IF st_config.b_config_fertig THEN
	(* Fehlermeldungen und Betriebsmeldungen ab dem Startindex in die globalen Meldungsarrays schreiben *)
	garr_stoermeldungen[st_config.i16_meld_startindex + 0] := sm_haspel_notaus;
	garr_stoermeldungen[st_config.i16_meld_startindex + 1] := sm_haspel_notabschaltung;
	garr_stoermeldungen[st_config.i16_meld_startindex + 2] := FALSE;
	garr_stoermeldungen[st_config.i16_meld_startindex + 3] := FALSE;
	garr_stoermeldungen[st_config.i16_meld_startindex + 4] := FALSE;
	garr_stoermeldungen[st_config.i16_meld_startindex + 5] := FALSE;
	garr_stoermeldungen[st_config.i16_meld_startindex + 6] := FALSE;
	garr_stoermeldungen[st_config.i16_meld_startindex + 7] := FALSE;
	garr_stoermeldungen[st_config.i16_meld_startindex + 8] := FALSE;
	garr_stoermeldungen[st_config.i16_meld_startindex + 9] := FALSE;
	garr_stoermeldungen[st_config.i16_meld_startindex + 10] := FALSE;
	garr_stoermeldungen[st_config.i16_meld_startindex + 11] := FALSE;
	garr_stoermeldungen[st_config.i16_meld_startindex + 12] := FALSE;
	garr_stoermeldungen[st_config.i16_meld_startindex + 13] := FALSE;
	garr_stoermeldungen[st_config.i16_meld_startindex + 14] := FALSE;
	garr_stoermeldungen[st_config.i16_meld_startindex + 15] := FALSE;
	garr_stoermeldungen[st_config.i16_meld_startindex + 16] := FALSE;
	garr_stoermeldungen[st_config.i16_meld_startindex + 17] := FALSE;
	garr_stoermeldungen[st_config.i16_meld_startindex + 18] := FALSE;
	garr_stoermeldungen[st_config.i16_meld_startindex + 19] := FALSE;
	
	garr_betriebsmeldungen[st_config.i16_meld_startindex + 0] := bm_haspel_bandende;
	garr_betriebsmeldungen[st_config.i16_meld_startindex + 1] := FALSE;
	garr_betriebsmeldungen[st_config.i16_meld_startindex + 2] := FALSE;
	garr_betriebsmeldungen[st_config.i16_meld_startindex + 3] := FALSE;
	garr_betriebsmeldungen[st_config.i16_meld_startindex + 4] := FALSE;
	garr_betriebsmeldungen[st_config.i16_meld_startindex + 5] := FALSE;
	garr_betriebsmeldungen[st_config.i16_meld_startindex + 6] := FALSE;
	garr_betriebsmeldungen[st_config.i16_meld_startindex + 7] := FALSE;
	garr_betriebsmeldungen[st_config.i16_meld_startindex + 8] := FALSE;
	garr_betriebsmeldungen[st_config.i16_meld_startindex + 9] := FALSE;
	garr_betriebsmeldungen[st_config.i16_meld_startindex + 10] := FALSE;
	garr_betriebsmeldungen[st_config.i16_meld_startindex + 11] := FALSE;
	garr_betriebsmeldungen[st_config.i16_meld_startindex + 12] := FALSE;
	garr_betriebsmeldungen[st_config.i16_meld_startindex + 13] := FALSE;
	garr_betriebsmeldungen[st_config.i16_meld_startindex + 14] := FALSE;
	garr_betriebsmeldungen[st_config.i16_meld_startindex + 15] := FALSE;
	garr_betriebsmeldungen[st_config.i16_meld_startindex + 16] := FALSE;
	garr_betriebsmeldungen[st_config.i16_meld_startindex + 17] := FALSE;
	garr_betriebsmeldungen[st_config.i16_meld_startindex + 18] := FALSE;
	garr_betriebsmeldungen[st_config.i16_meld_startindex + 19] := FALSE;
END_IF
END_FUNCTION_BLOCK

(* POU Gemeinsamkeiten17xx/Oeler/ST_Bandoeler, ST *)
FUNCTION_BLOCK ST_Bandoeler
VAR_INPUT
	st_config						: struct_config;
	st_ctrl_in						: struct_ctrl_in;
	b_ot_spur					: BOOL;
END_VAR
VAR_IN_OUT
	st_daten						: struct_oeler_daten;
	st_visu						: struct_oeler_visu;
END_VAR
VAR_OUTPUT
	st_ctrl_out					: struct_ctrl_out;
END_VAR
VAR
	fb_ton_quitt					: TON;
	dt_datum_uhrzeit_letzte_oelung	: DT;
	fb_state_entry					: ST_StateEntry;
	t_delta_zeitraum				: TIME := t#5h;
	t_blaszeit					: TIME := t#500ms;
	fb_ton_oelzeit					: TON;
	fb_ton_blaszeit				: TON;
	fb_r_trig_start_oelen			: R_TRIG;
	fb_r_trig_hubimpuls			: R_TRIG;
	i32_default_wert_intervall		: INT := 1000;

	fb_r_trig_ibn_handoelen		: R_TRIG;
	fb_ton_ibn_handoelen			: TON;
	b_ibn_handoelen				: BOOL := FALSE;

	a_ventil_oel		 			AT %Q* : BOOL;
	a_ventil_luft		 			AT %Q* : BOOL;
END_VAR
(* Bandöler mit Zwangs- und Stillstandsölung *)
(* Oeler Impuls generieren *)
fb_ton_oelzeit(IN:= , PT:= , Q=> , ET=> );
fb_ton_blaszeit(IN:= , PT:= t_blaszeit, Q=> , ET=> );
fb_ton_quitt(IN:= , PT:= t#100ms, Q=> , ET=> );

(* Hubimpuls *)
fb_r_trig_hubimpuls(CLK:= b_ot_spur, Q=> );

(* Inbetriebnahme *)
fb_r_trig_ibn_handoelen(CLK:= b_ibn_handoelen, Q=> );
fb_ton_ibn_handoelen(IN:= , PT:= t#1s, Q=> , ET=> );
IF fb_r_trig_ibn_handoelen.Q THEN
	fb_ton_ibn_handoelen.IN := TRUE;
ELSE
	IF fb_ton_ibn_handoelen.Q THEN
		b_ibn_handoelen := FALSE;
	 	fb_ton_ibn_handoelen.IN := FALSE;
	END_IF
END_IF

(* =======================================Toplevel========================================== *)
IF fb_state_entry.i16_next_step > INIT AND fb_state_entry.i16_next_step < FEHLER THEN
	IF fb_state_entry.i16_next_step < STOP THEN
		IF st_ctrl_in.b_stop THEN
			fb_state_entry.i16_next_step := STOP;
		END_IF
	END_IF
END_IF

(* Prüfe auf neue Intervalvorgabe *)
IF st_config.b_station_aktiv AND st_daten.i32_neue_intervallvorgabe <> st_daten.i32_alte_intervallvorgabe THEN
	st_daten.i32_alte_intervallvorgabe := st_daten.i32_neue_intervallvorgabe;
	st_daten.i32_aktueller_stand := st_daten.i32_neue_intervallvorgabe;
END_IF

(* Zähle Hübe *)
IF st_config.b_station_aktiv AND fb_r_trig_hubimpuls.Q THEN
	(* Von der Intervallvorgabe wird runter gezählt bis Null. Dann kommt der Ölimpuls *)
	st_daten.i32_aktueller_stand := st_daten.i32_aktueller_stand - 1;
END_IF

(* ==================================Schrittkette================================ *)
fb_state_entry(
	i16_next_step:= , 
	i16_pos:= 1,
	s_debugtext:= ,
	E=> ,
	X=> , 
	i16_step=> ,
	i16_last_step=> );

CASE fb_state_entry.i16_step OF
(*=======================================================*)
	INIT_OBJ:
		IF st_config.b_config_fertig THEN
			fb_state_entry.i16_next_step := INIT;
		END_IF
		
(*=======================================================*)
	INIT:
		IF fb_state_entry.E THEN
			fb_ton_blaszeit.IN := FALSE;
			fb_ton_oelzeit.IN := FALSE;
			st_ctrl_out.b_fehler := FALSE;
			st_ctrl_out.b_bereit := FALSE;
			st_ctrl_out.b_fertig := FALSE;
			a_ventil_oel := FALSE;
			a_ventil_luft := FALSE;
		END_IF

		(*-----------------------Weiterschaltbedingungen----------------------------*)
		IF st_ctrl_in.b_init THEN
			IF st_config.b_station_aktiv THEN
				fb_state_entry.i16_next_step := 20;
			ELSE
				fb_state_entry.i16_next_step := BEREIT;
			END_IF
		END_IF

(*=======================================================*)
	20: (* Abfrage Datum / Uhrzeit wegen Ölen nach Stillstand*)

		(*-----------------------Weiterschaltbedingungen----------------------------*)
		IF (gdt_system_time - dt_datum_uhrzeit_letzte_oelung) > t_delta_zeitraum THEN
			fb_ton_oelzeit.PT := st_daten.t_oelzeit_nach_stillstand;
			fb_state_entry.i16_next_step := 110;
		ELSE
			fb_state_entry.i16_next_step := BEREIT;
		END_IF

(*=======================================================*)
	BEREIT:
		IF fb_state_entry.E THEN
			st_ctrl_out.b_bereit := TRUE;
		END_IF

		(*-----------------------Weiterschaltbedingungen----------------------------*)
		IF  st_config.b_station_aktiv AND (st_daten.i32_aktueller_stand <= 0 OR st_visu.b_handoelen OR fb_r_trig_ibn_handoelen.Q) THEN
			st_visu.b_handoelen := FALSE;
			fb_ton_oelzeit.PT := st_daten.t_ventiloeffnungszeit;
			fb_state_entry.i16_next_step := 110;
		END_IF

(*=======================================================*)
	110: (* Luft einschalten *)
		IF fb_state_entry.E THEN
			fb_ton_blaszeit.IN := TRUE;
			a_ventil_luft := TRUE;
		END_IF

		(*-----------------------Weiterschaltbedingungen----------------------------*)
		IF  fb_ton_blaszeit.Q THEN
			fb_ton_blaszeit.IN := FALSE;
			fb_state_entry.i16_next_step := 120;
		END_IF

(*=======================================================*)
	120: (* Ölen *)
		IF fb_state_entry.E THEN
			dt_datum_uhrzeit_letzte_oelung := gdt_system_time;	(* Merken wann das letze mal geölt wurde *)
			IF st_daten.i32_neue_intervallvorgabe <= 0 THEN
				 st_daten.i32_neue_intervallvorgabe := i32_default_wert_intervall;	(* Verhindere Dauerölung, wenn in den WKZ-Ölerdaten noch 0 drin steht *)
			END_IF
			st_daten.i32_aktueller_stand := st_daten.i32_neue_intervallvorgabe;
			fb_ton_oelzeit.IN := TRUE;
			a_ventil_oel := TRUE;
		END_IF

		(*-----------------------Weiterschaltbedingungen----------------------------*)
		IF  fb_ton_oelzeit.Q THEN
			fb_ton_oelzeit.IN := FALSE;
			a_ventil_oel := FALSE;
			a_ventil_luft := FALSE;
			fb_state_entry.i16_next_step := BEREIT;
		END_IF

(*=======================================================*)
	FEHLER:
		IF fb_state_entry.E THEN
			st_ctrl_out.b_fehler := TRUE;
			a_ventil_oel := FALSE;
			a_ventil_luft := FALSE;
			fb_ton_quitt.IN := FALSE;
		END_IF

		(*-----------------------Weiterschaltbedingungen----------------------------*)
		IF st_ctrl_in.b_quitt AND NOT fb_state_entry.E THEN
			st_ctrl_out.b_fehler := FALSE;
			fb_ton_quitt.IN := TRUE;
		END_IF

		IF fb_ton_quitt.Q THEN
			fb_ton_quitt.IN := FALSE;
			fb_state_entry.i16_next_step := INIT;
		END_IF

(*=======================================================*)
	STOP:
		IF fb_state_entry.E THEN
			a_ventil_oel := FALSE;
			a_ventil_luft := FALSE;
			fb_ton_quitt.IN := FALSE;
		END_IF

		(*-----------------------Weiterschaltbedingungen----------------------------*)
		IF st_ctrl_in.b_quitt AND NOT fb_state_entry.E THEN
			fb_ton_quitt.IN := TRUE;
		END_IF

		IF fb_ton_quitt.Q THEN
			fb_ton_quitt.IN := FALSE;
			fb_state_entry.i16_next_step := INIT;
		END_IF
END_CASE

fb_state_entry(
	i16_next_step:= , 
	i16_pos:= 2,
	s_debugtext:= ,
	E=> ,
	X=> , 
	i16_step=> ,
	i16_last_step=> );

IF st_config.b_config_fertig THEN
	(* Fehlermeldungen und Betriebsmeldungen ab dem Startindex in die globalen Meldungsarrays schreiben *)
	garr_stoermeldungen[st_config.i16_meld_startindex + 0] := FALSE;
	garr_stoermeldungen[st_config.i16_meld_startindex + 1] := FALSE;
	garr_stoermeldungen[st_config.i16_meld_startindex + 2] := FALSE;
	garr_stoermeldungen[st_config.i16_meld_startindex + 3] := FALSE;
	garr_stoermeldungen[st_config.i16_meld_startindex + 4] := FALSE;
	garr_stoermeldungen[st_config.i16_meld_startindex + 5] := FALSE;
	garr_stoermeldungen[st_config.i16_meld_startindex + 6] := FALSE;
	garr_stoermeldungen[st_config.i16_meld_startindex + 7] := FALSE;
	garr_stoermeldungen[st_config.i16_meld_startindex + 8] := FALSE;
	garr_stoermeldungen[st_config.i16_meld_startindex + 9] := FALSE;
	garr_stoermeldungen[st_config.i16_meld_startindex + 10] := FALSE;
	garr_stoermeldungen[st_config.i16_meld_startindex + 11] := FALSE;
	garr_stoermeldungen[st_config.i16_meld_startindex + 12] := FALSE;
	garr_stoermeldungen[st_config.i16_meld_startindex + 13] := FALSE;
	garr_stoermeldungen[st_config.i16_meld_startindex + 14] := FALSE;
	garr_stoermeldungen[st_config.i16_meld_startindex + 15] := FALSE;
	garr_stoermeldungen[st_config.i16_meld_startindex + 16] := FALSE;
	garr_stoermeldungen[st_config.i16_meld_startindex + 17] := FALSE;
	garr_stoermeldungen[st_config.i16_meld_startindex + 18] := FALSE;
	garr_stoermeldungen[st_config.i16_meld_startindex + 19] := FALSE;
	
	garr_betriebsmeldungen[st_config.i16_meld_startindex + 0] := FALSE;
	garr_betriebsmeldungen[st_config.i16_meld_startindex + 1] := FALSE;
	garr_betriebsmeldungen[st_config.i16_meld_startindex + 2] := FALSE;
	garr_betriebsmeldungen[st_config.i16_meld_startindex + 3] := FALSE;
	garr_betriebsmeldungen[st_config.i16_meld_startindex + 4] := FALSE;
	garr_betriebsmeldungen[st_config.i16_meld_startindex + 5] := FALSE;
	garr_betriebsmeldungen[st_config.i16_meld_startindex + 6] := FALSE;
	garr_betriebsmeldungen[st_config.i16_meld_startindex + 7] := FALSE;
	garr_betriebsmeldungen[st_config.i16_meld_startindex + 8] := FALSE;
	garr_betriebsmeldungen[st_config.i16_meld_startindex + 9] := FALSE;
	garr_betriebsmeldungen[st_config.i16_meld_startindex + 10] := FALSE;
	garr_betriebsmeldungen[st_config.i16_meld_startindex + 11] := FALSE;
	garr_betriebsmeldungen[st_config.i16_meld_startindex + 12] := FALSE;
	garr_betriebsmeldungen[st_config.i16_meld_startindex + 13] := FALSE;
	garr_betriebsmeldungen[st_config.i16_meld_startindex + 14] := FALSE;
	garr_betriebsmeldungen[st_config.i16_meld_startindex + 15] := FALSE;
	garr_betriebsmeldungen[st_config.i16_meld_startindex + 16] := FALSE;
	garr_betriebsmeldungen[st_config.i16_meld_startindex + 17] := FALSE;
	garr_betriebsmeldungen[st_config.i16_meld_startindex + 18] := FALSE;
	garr_betriebsmeldungen[st_config.i16_meld_startindex + 19] := FALSE;
END_IF
END_FUNCTION_BLOCK

(* POU Gemeinsamkeiten17xx/Stueckzahlen/ST_Stueckzahl, ST *)
FUNCTION_BLOCK ST_Stueckzahl
VAR_INPUT
	b_wkz_zweifachfallend			: BOOL;
	st_config						: struct_config;
	st_ctrl_in						: struct_ctrl_in;
END_VAR
VAR_OUTPUT
	st_ctrl_out					: struct_ctrl_out;
END_VAR
VAR
	fb_ton_wz					: TON;
	fb_ton_uez					: TON;
	fb_ton_quitt					: TON;
	fb_r_trig_gutteil				: R_TRIG;
	fb_r_trig_schlechtteil			: R_TRIG;
	fb_state_entry					: ST_StateEntry;
	i							: INT;
	sm_auftrag_voll				: BOOL := FALSE;
	sm_verpackungseinheit_voll	: BOOL := FALSE;
	i16_faktor_wkz				: INT := 1;
END_VAR
(* Zeiten *)
fb_ton_wz(IN:= , PT:= , Q=>  , ET=> );
fb_ton_uez(IN:= , PT:= , Q=>  , ET=> );
fb_ton_quitt(IN:= , PT:= t#100ms, Q=> , ET=> );

(* Flanken *)
fb_r_trig_gutteil(CLK:= st_ctrl_in.b_gutteil_produziert, Q=> );
fb_r_trig_schlechtteil(CLK:= st_ctrl_in.b_schlechtteil_produziert, Q=> );


IF b_wkz_zweifachfallend THEN
	i16_faktor_wkz := 2;
ELSE
	i16_faktor_wkz := 1;
END_IF

(* Toplevel *)
IF fb_state_entry.i16_next_step > INIT AND fb_state_entry.i16_next_step < FEHLER THEN
	IF fb_state_entry.i16_next_step < STOP THEN
		IF st_ctrl_in.b_stop THEN
			fb_state_entry.i16_next_step := STOP;
		END_IF
	END_IF

	(* Zählerstände rücksetzen *)
	FOR i := 0 TO (SIZEOF (gst_datensatz.st_stueckzahlen.st_teilezaehler) / SIZEOF (gst_datensatz.st_stueckzahlen.st_teilezaehler[0])) - 1  BY 1 DO
		IF gst_datensatz.st_stueckzahlen.st_teilezaehler[i].b_reset_gutteile THEN
			gst_datensatz.st_stueckzahlen.st_teilezaehler[i].i32_aktuelle_gutteile := 0;
		END_IF
		IF gst_datensatz.st_stueckzahlen.st_teilezaehler[i].b_reset_schlechtteile THEN
			gst_datensatz.st_stueckzahlen.st_teilezaehler[i].i32_aktuelle_schlechtteile := 0;
		END_IF
	END_FOR
END_IF

(* ==================================Schrittkette================================ *)
fb_state_entry(
	i16_next_step:= , 
	i16_pos:= 1,
	s_debugtext:= ,
	E=> ,
	X=> , 
	i16_step=> ,
	i16_last_step=> );

CASE fb_state_entry.i16_step OF
(*=======================================================*)
	INIT_OBJ:
		IF st_config.b_config_fertig THEN
			fb_state_entry.i16_next_step := INIT;
		END_IF

(*=======================================================*)
	INIT:
		IF fb_state_entry.E THEN
			fb_ton_wz.IN := FALSE;
			fb_ton_uez.IN := FALSE;
			fb_ton_quitt.IN := FALSE;
			sm_auftrag_voll := FALSE;
			sm_verpackungseinheit_voll := FALSE;
			st_ctrl_out.b_fehler := FALSE;
			st_ctrl_out.b_bereit := FALSE;
			st_ctrl_out.b_fertig := FALSE;
		END_IF

		(*-----------------------Weiterschaltbedingungen----------------------------*)
		IF st_ctrl_in.b_init THEN
			fb_state_entry.i16_next_step := BEREIT;
		END_IF

(*=======================================================*)
	BEREIT:
		IF fb_state_entry.E THEN
			st_ctrl_out.b_bereit := TRUE;
		END_IF

		(* Zähler hochzählen *)
		IF fb_r_trig_gutteil.Q THEN
			gst_datensatz.st_stueckzahlen.st_teilezaehler[JAHR].i32_aktuelle_gutteile := gst_datensatz.st_stueckzahlen.st_teilezaehler[JAHR].i32_aktuelle_gutteile + i16_faktor_wkz;
			gst_datensatz.st_stueckzahlen.st_teilezaehler[VPE].i32_aktuelle_gutteile := gst_datensatz.st_stueckzahlen.st_teilezaehler[VPE].i32_aktuelle_gutteile + i16_faktor_wkz;
		END_IF

		IF fb_r_trig_schlechtteil.Q THEN
			gst_datensatz.st_stueckzahlen.st_teilezaehler[JAHR].i32_aktuelle_schlechtteile := gst_datensatz.st_stueckzahlen.st_teilezaehler[JAHR].i32_aktuelle_schlechtteile + i16_faktor_wkz;
			gst_datensatz.st_stueckzahlen.st_teilezaehler[VPE].i32_aktuelle_schlechtteile := gst_datensatz.st_stueckzahlen.st_teilezaehler[VPE].i32_aktuelle_schlechtteile + i16_faktor_wkz;
		END_IF

		(* Eine Verpackungseinheit ist voll *)
		IF 	gst_datensatz.st_stueckzahlen.st_teilezaehler[VPE].i32_aktuelle_gutteile >= gst_datensatz.st_stueckzahlen.st_teilezaehler[VPE].i32_vorgabe_gutteile AND
			fb_state_entry.i16_next_step <> FEHLER
			THEN
				gst_datensatz.st_stueckzahlen.st_teilezaehler[AUFTRAG].i32_aktuelle_gutteile := gst_datensatz.st_stueckzahlen.st_teilezaehler[AUFTRAG].i32_aktuelle_gutteile + 1;
				sm_verpackungseinheit_voll := TRUE;
				fb_state_entry.i16_next_step := FEHLER;
		END_IF
		(* Gesamter Auftrag ist voll *)
		IF 	gst_datensatz.st_stueckzahlen.st_teilezaehler[AUFTRAG].i32_aktuelle_gutteile >= gst_datensatz.st_stueckzahlen.st_teilezaehler[AUFTRAG].i32_vorgabe_gutteile AND
			fb_state_entry.i16_next_step <> FEHLER
			THEN
				sm_auftrag_voll := TRUE;
				fb_state_entry.i16_next_step := FEHLER;
		END_IF

(*=======================================================*)
	FEHLER:
		IF fb_state_entry.E THEN
			st_ctrl_out.b_fehler := TRUE;
		END_IF

		(*-----------------------Weiterschaltbedingungen----------------------------*)
		IF st_ctrl_in.b_quitt AND NOT fb_state_entry.E THEN
			st_ctrl_out.b_fehler := FALSE;
			fb_ton_quitt.IN := TRUE;

			IF gst_datensatz.st_stueckzahlen.st_teilezaehler[VPE].i32_aktuelle_gutteile >= gst_datensatz.st_stueckzahlen.st_teilezaehler[VPE].i32_vorgabe_gutteile THEN
				gst_datensatz.st_stueckzahlen.st_teilezaehler[VPE].i32_aktuelle_gutteile := 0;
				sm_verpackungseinheit_voll := FALSE;
			END_IF
			IF gst_datensatz.st_stueckzahlen.st_teilezaehler[AUFTRAG].i32_aktuelle_gutteile >= gst_datensatz.st_stueckzahlen.st_teilezaehler[AUFTRAG].i32_vorgabe_gutteile THEN
				gst_datensatz.st_stueckzahlen.st_teilezaehler[AUFTRAG].i32_aktuelle_gutteile := 0;
				sm_auftrag_voll := FALSE;
			END_IF
		END_IF

		IF fb_ton_quitt.Q THEN
			fb_ton_quitt.IN := FALSE;
			fb_state_entry.i16_next_step := INIT;
		END_IF

(*=======================================================*)
	STOP:

		(*-----------------------Weiterschaltbedingungen----------------------------*)
		IF st_ctrl_in.b_quitt AND NOT fb_state_entry.E THEN
			fb_ton_quitt.IN := TRUE;
		END_IF

		IF fb_ton_quitt.Q THEN
			fb_ton_quitt.IN := FALSE;
			fb_state_entry.i16_next_step := INIT;
		END_IF
END_CASE

fb_state_entry(
	i16_next_step:= , 
	i16_pos:= 2,
	s_debugtext:= ,
	E=> , 
	X=> , 
	i16_step=> ,
	i16_last_step=> );

IF st_config.b_config_fertig THEN
	(* Fehlermeldungen und Betriebsmeldungen ab dem Startindex in die globalen Meldungsarrays schreiben *)
	garr_stoermeldungen[st_config.i16_meld_startindex + 0] := sm_verpackungseinheit_voll;
	garr_stoermeldungen[st_config.i16_meld_startindex + 1] := sm_auftrag_voll;
	garr_stoermeldungen[st_config.i16_meld_startindex + 2] := FALSE;
	garr_stoermeldungen[st_config.i16_meld_startindex + 3] := FALSE;
	garr_stoermeldungen[st_config.i16_meld_startindex + 4] := FALSE;
	garr_stoermeldungen[st_config.i16_meld_startindex + 5] := FALSE;
	garr_stoermeldungen[st_config.i16_meld_startindex + 6] := FALSE;
	garr_stoermeldungen[st_config.i16_meld_startindex + 7] := FALSE;
	garr_stoermeldungen[st_config.i16_meld_startindex + 8] := FALSE;
	garr_stoermeldungen[st_config.i16_meld_startindex + 9] := FALSE;
	garr_stoermeldungen[st_config.i16_meld_startindex + 10] := FALSE;
	garr_stoermeldungen[st_config.i16_meld_startindex + 11] := FALSE;
	garr_stoermeldungen[st_config.i16_meld_startindex + 12] := FALSE;
	garr_stoermeldungen[st_config.i16_meld_startindex + 13] := FALSE;
	garr_stoermeldungen[st_config.i16_meld_startindex + 14] := FALSE;
	garr_stoermeldungen[st_config.i16_meld_startindex + 15] := FALSE;
	garr_stoermeldungen[st_config.i16_meld_startindex + 16] := FALSE;
	garr_stoermeldungen[st_config.i16_meld_startindex + 17] := FALSE;
	garr_stoermeldungen[st_config.i16_meld_startindex + 18] := FALSE;
	garr_stoermeldungen[st_config.i16_meld_startindex + 19] := FALSE;
	
	garr_betriebsmeldungen[st_config.i16_meld_startindex + 0] := FALSE;
	garr_betriebsmeldungen[st_config.i16_meld_startindex + 1] := FALSE;
	garr_betriebsmeldungen[st_config.i16_meld_startindex + 2] := FALSE;
	garr_betriebsmeldungen[st_config.i16_meld_startindex + 3] := FALSE;
	garr_betriebsmeldungen[st_config.i16_meld_startindex + 4] := FALSE;
	garr_betriebsmeldungen[st_config.i16_meld_startindex + 5] := FALSE;
	garr_betriebsmeldungen[st_config.i16_meld_startindex + 6] := FALSE;
	garr_betriebsmeldungen[st_config.i16_meld_startindex + 7] := FALSE;
	garr_betriebsmeldungen[st_config.i16_meld_startindex + 8] := FALSE;
	garr_betriebsmeldungen[st_config.i16_meld_startindex + 9] := FALSE;
	garr_betriebsmeldungen[st_config.i16_meld_startindex + 10] := FALSE;
	garr_betriebsmeldungen[st_config.i16_meld_startindex + 11] := FALSE;
	garr_betriebsmeldungen[st_config.i16_meld_startindex + 12] := FALSE;
	garr_betriebsmeldungen[st_config.i16_meld_startindex + 13] := FALSE;
	garr_betriebsmeldungen[st_config.i16_meld_startindex + 14] := FALSE;
	garr_betriebsmeldungen[st_config.i16_meld_startindex + 15] := FALSE;
	garr_betriebsmeldungen[st_config.i16_meld_startindex + 16] := FALSE;
	garr_betriebsmeldungen[st_config.i16_meld_startindex + 17] := FALSE;
	garr_betriebsmeldungen[st_config.i16_meld_startindex + 18] := FALSE;
	garr_betriebsmeldungen[st_config.i16_meld_startindex + 19] := FALSE;
END_IF
END_FUNCTION_BLOCK

(* POU Gemeinsamkeiten17xx/XML Server/FB_2OrdnerMitDateiErstellen, ST *)
FUNCTION_BLOCK FB_2OrdnerMitDateiErstellen
VAR_INPUT
	bExecute					: BOOL;
	bQuit						: BOOL;
	s_path						: STRING;
	s_dateiname					: STRING;
	s_datei_erweiterung			: STRING;
	s_x_path_name				: STRING;
	s_symname					: STRING;
END_VAR
VAR_IN_OUT
END_VAR
VAR_OUTPUT
	bBusy						: BOOL;
	bError						: BOOL;
	nErrId						: UDINT;

END_VAR
VAR
	fb_enum_find_file_list			: FB_EnumFindFileList;
	fb_enum_find_file_entry			: FB_EnumFindFileEntry;
	fb_create_directory			: FB_CreateDir;	(* mit diesem FB kan nur eine Ordnerverzeichnissstruktur angelegt werden, jedoch keine Dateien erzeugt werden *)
	fb_file_open					: FB_FileOpen;	(* Eine vorhandene Datei öffnen oder eine Neue erzeugen *)
	fb_file_close					: FB_FileClose;
	fb_file_write					: FB_FileWrite;
	h_filehandle					: UINT := 0;(* file handle of the file *)
	arr_file_list					: ARRAY[0..63] OF ST_FindFileEntry;
	fb_ton_quitt					: TON;
	fb_r_trig_execute				: R_TRIG;
	fb_state_entry					: ST_StateEntry;
	temp_string					: STRING[255];
	i16_file_entry_zaehler			: INT := 0;
	i16_file_nr					: INT := 0;
	i							: INT := 0;
	b_pfad_vorhanden			: BOOL;
	b_datei_vorhanden			: BOOL;
	arr_rootpath					: ARRAY[0..2] OF STRING;
END_VAR
fb_r_trig_execute(CLK:= bExecute, Q=> );
fb_ton_quitt(IN:= , PT:= t#100ms, Q=> , ET=> );

(* ======================================Schrittkette======================================== *)
fb_state_entry(
	i16_next_step:= ,
	i16_pos:= 1,
	s_debugtext:= ,
	E=> ,
	X=> ,
	i16_step=> ,
	i16_last_step=> );

CASE fb_state_entry.i16_step OF
(*=======================================================*)
	0:(* INIT *)
		bBusy := FALSE;
		bError := FALSE;
		nErrId := 0;
		fb_create_directory.bExecute := FALSE;
		fb_enum_find_file_list.bExecute := FALSE;
		fb_enum_find_file_entry.bExecute := FALSE;
		fb_file_open.bExecute := FALSE;
		fb_file_close.bExecute := FALSE;
		fb_state_entry.i16_next_step := 10;

(*=======================================================*)
	10:	(* Warte auf Execute-Befehl *)
		IF fb_state_entry.E THEN
			bBusy := FALSE;
		END_IF

		IF fb_r_trig_execute.Q THEN
			bBusy := TRUE;
			b_pfad_vorhanden := FALSE;
			b_datei_vorhanden := FALSE;
			arr_rootpath[0] := MID(s_path, 1,3);
			arr_rootpath[1] := MID(s_path, 4,3);
			arr_rootpath[2] := MID(s_path, 10,3);
			fb_state_entry.i16_next_step := 20;
		END_IF

(*=======================================================*)
	20:	(* Prüfe, ob gewünschter Pfad auf dem Maschinen-PC vorhanden ist *)
		IF fb_state_entry.E THEN
			fb_enum_find_file_list.sPathName := s_path;
			fb_enum_find_file_list.eCmd := eEnumCmd_First;
			fb_enum_find_file_list.bExecute := TRUE;
		END_IF

		IF fb_enum_find_file_list.bBusy THEN
			fb_enum_find_file_list.bExecute := FALSE;
			fb_state_entry.i16_next_step := 30;
		END_IF

(*=======================================================*)
	30:	(* Auswerten des Ordner-Suchergebnis *)
		IF NOT fb_enum_find_file_list.bBusy THEN
			fb_enum_find_file_list.bExecute := FALSE;
		 	IF fb_enum_find_file_list.bError OR fb_enum_find_file_list.bEOE THEN
				 IF fb_enum_find_file_list.nFindFiles=0 THEN
					b_pfad_vorhanden := FALSE;
					fb_state_entry.i16_next_step := 40;	(* Pfad nicht vorhanden -> wird angelegt *)
				ELSE
					b_pfad_vorhanden := TRUE;
					fb_state_entry.i16_next_step := 60;	(* O.K. Pfad vorhanden -> Datei prüfen *)
				END_IF
			END_IF
		END_IF

(*=======================================================*)
	40:	(* Erstellen des ersten Ordnerverzeichnisses auf dem Laufwerk des Maschinen-PCs *)
		IF fb_state_entry.E THEN
			fb_create_directory.sPathName := s_path;
			fb_create_directory.bExecute := TRUE;
		END_IF

		IF fb_create_directory.bBusy THEN
			fb_create_directory.bExecute := FALSE;
			fb_state_entry.i16_next_step := 50;
		END_IF

(*=======================================================*)
	50:	(* Ordner wurde erstellt *)
		IF NOT fb_create_directory.bBusy  THEN
			IF NOT fb_create_directory.bError THEN
				fb_state_entry.i16_next_step := 60;	(* Ordnerverzeichnis wurde erfolgreich erstellt -> eine neue Datei anlegen oder eine Vorhandene öffnen *)
			ELSE
				fb_state_entry.i16_next_step := 1000;	(* Fehler *)
			END_IF
		END_IF

(*=======================================================*)
	60:	(* Prüfe, ob die gewünschte Datei in diesem Ordnerverzeichnis vorhanden ist *)
		IF fb_state_entry.E THEN
			temp_string := '';
			temp_string := CONCAT(temp_string, s_path);
			temp_string := CONCAT(temp_string, '\');
			temp_string := CONCAT(temp_string, s_dateiname);
			temp_string := CONCAT(temp_string, s_datei_erweiterung);
			fb_enum_find_file_entry.sPathName := temp_string;
			fb_enum_find_file_entry.eCmd := eEnumCmd_First;
			fb_enum_find_file_entry.bExecute := TRUE;
		END_IF

		IF fb_enum_find_file_entry.bBusy THEN
			fb_enum_find_file_entry.bExecute := FALSE;
			fb_state_entry.i16_next_step := 70;
		END_IF

(*=======================================================*)
	70:	(* Auswerten des Datei-Suchergebnis *)
		IF NOT fb_enum_find_file_entry.bBusy THEN
			fb_enum_find_file_entry.bExecute := FALSE;
		 	IF NOT fb_enum_find_file_entry.bError THEN
				IF fb_enum_find_file_entry.bEOE THEN
					IF fb_enum_find_file_entry.stFindFile.sFileName = CONCAT(s_dateiname, s_datei_erweiterung) THEN
					(* Datei bereits vorhanden *)
						b_datei_vorhanden := TRUE;
						fb_state_entry.i16_next_step := 0;
					ELSE
					(* Ende der Fileliste wurde erreicht und die gesuchte Datei ist  nicht vorhanden -> muss später angelegt werden *)
						b_datei_vorhanden := FALSE;
						fb_state_entry.i16_next_step := 100;
					END_IF
				ELSE
				(* Dateisuche im FB mit Abort korrekt beenden *)
					IF fb_enum_find_file_entry.stFindFile.sFileName = CONCAT(s_dateiname, s_datei_erweiterung) THEN
					(* Die gesuchte Datei wurde in der Fileliste gefunden *)
						b_datei_vorhanden := TRUE;
						fb_state_entry.i16_next_step := 80;
					ELSE
					(* Datei ist  nicht vorhanden -> muss später angelegt werden *)
						b_datei_vorhanden := FALSE;
						fb_state_entry.i16_next_step := 80;
					END_IF
				END_IF
			ELSE
				fb_state_entry.i16_next_step := FEHLER;
			END_IF
		END_IF

(*=======================================================*)
	80:	(* Dateisuchen wird beendet *)
		IF fb_state_entry.E THEN
			fb_enum_find_file_entry.eCmd := eEnumCmd_Abort;
			fb_enum_find_file_entry.bExecute := TRUE;
		END_IF

		IF fb_enum_find_file_entry.bBusy THEN
			fb_enum_find_file_entry.bExecute := FALSE;
			fb_state_entry.i16_next_step := 90;
		END_IF

(*=======================================================*)
	90:	(* Filehandle wieder frei *)
		IF NOT fb_enum_find_file_entry.bBusy THEN
			fb_enum_find_file_entry.bExecute := FALSE;
		 	IF NOT fb_enum_find_file_entry.bError AND fb_enum_find_file_entry.bEOE THEN
				fb_state_entry.i16_next_step := 100;
			ELSE
				fb_state_entry.i16_next_step := FEHLER;
			END_IF
		END_IF

(*=======================================================*)
	100:	(* Abfrage auf Datei anlegen *)
		IF fb_state_entry.E THEN
			IF NOT b_datei_vorhanden THEN
				fb_state_entry.i16_next_step := 110;
			ELSE
				fb_state_entry.i16_next_step := 0;	(* Fertig *)
			END_IF
		END_IF

(*=======================================================*)
	110:	(* Erzeugen einer neuen Datei *)
		IF fb_state_entry.E THEN
			temp_string := '';
			temp_string := CONCAT(temp_string, s_path);
			temp_string := CONCAT(temp_string, '\');
			temp_string := CONCAT(temp_string, s_dateiname);
			temp_string := CONCAT(temp_string, s_datei_erweiterung);
			fb_file_open.sPathName := temp_string;
			fb_file_open.nMode := FOPEN_MODEWRITE OR FOPEN_MODEBINARY;
			fb_file_open.bExecute := TRUE;
		END_IF

		IF fb_file_open.bBusy THEN
			fb_file_open.bExecute := FALSE;
			fb_state_entry.i16_next_step := 120;
		END_IF

(*=======================================================*)
	120:	(* Warte bis Datei geöffnet wurde *)
		IF NOT fb_file_open.bBusy  THEN
			IF NOT fb_file_open.bError THEN
				h_filehandle := fb_file_open.hFile;
				fb_state_entry.i16_next_step := 130;
			ELSE	(* Fehler *)
				nErrId := fb_file_open.nErrId;
				fb_state_entry.i16_next_step := 1000;
			END_IF
		END_IF

(*=======================================================*)
	130:	(* Schreibe die Dateistruktur im XML-Format: z.B.*)
		(*
		<Maschine1700_Datensicherung>
		<gst_datensatz>
		</gst_datensatz>
		</Maschine1700_Datensicherung>
		*)
		IF fb_state_entry.E THEN
			temp_string := '';
			temp_string := CONCAT(temp_string, '<');
			temp_string := CONCAT(temp_string, s_x_path_name);
			temp_string := CONCAT(temp_string, '>');
			temp_string := CONCAT(temp_string, '$r$n');

			(* Die Variable "s_xml_variablenname" wird hier schon mit angelegt, *)
			(* damit später beim "WECHSELN>" daraus gelesen werden kann, obwohl noch nichts drin steht *)
			temp_string := CONCAT(temp_string, '<');
			temp_string := CONCAT(temp_string, s_symname);
			temp_string := CONCAT(temp_string, '>');
			temp_string := CONCAT(temp_string, '$r$n');
			temp_string := CONCAT(temp_string, '<');
			temp_string := CONCAT(temp_string, '/');
			temp_string := CONCAT(temp_string, s_symname);
			temp_string := CONCAT(temp_string, '>');
			temp_string := CONCAT(temp_string, '$r$n');

			temp_string := CONCAT(temp_string, '<');
			temp_string := CONCAT(temp_string, '/');
			temp_string := CONCAT(temp_string, s_x_path_name);
			temp_string := CONCAT(temp_string, '>');
			fb_file_write.hFile := h_filehandle;
 			fb_file_write.bExecute := TRUE;
		END_IF

		IF fb_file_write.bBusy THEN
			fb_file_write.bExecute := FALSE;
			fb_state_entry.i16_next_step := 140;
		END_IF

(*=======================================================*)
	140:	(* Warte bis Datei geschrieben wurde *)
		IF NOT fb_file_write.bBusy  THEN
			IF NOT fb_file_write.bError THEN
				fb_state_entry.i16_next_step := 150;
			ELSE	(* Fehler *)
				nErrId := fb_file_write.nErrId;
				fb_state_entry.i16_next_step := 1000;
			END_IF
		END_IF

(*=======================================================*)
	150:	(* Schliesse Datei wieder, damit ein erneuter Zugriff möglich ist *)
		IF fb_state_entry.E THEN
			fb_file_close.hFile := h_filehandle;
			fb_file_close.bExecute := TRUE;
		END_IF

		IF fb_file_close.bBusy THEN
			fb_file_close.bExecute := FALSE;
			fb_state_entry.i16_next_step := 160;
		END_IF

(*=======================================================*)
	160:	(* Warte bis geschlossen *)
		IF NOT fb_file_close.bBusy  THEN
			IF NOT fb_file_close.bError THEN
				h_filehandle := 0;
				fb_state_entry.i16_next_step :=0;
			ELSE	(* Fehler *)
				nErrId := fb_file_close.nErrId;
				fb_state_entry.i16_next_step := 1000;
			END_IF
		END_IF

(*=======================================================*)
	1000: (* Fehler *)
		IF fb_state_entry.E THEN
			bBusy := FALSE;
			bError := TRUE;
			fb_ton_quitt.IN := FALSE;
		END_IF

		(*-----------------------Weiterschaltbedingungen----------------------------*)
		IF bQuit AND NOT fb_state_entry.E THEN
			bError := FALSE;
			fb_ton_quitt.IN := TRUE;
		END_IF

		IF fb_ton_quitt.Q THEN
			fb_ton_quitt.IN := FALSE;
			fb_state_entry.i16_next_step := 0;
		END_IF
END_CASE

fb_state_entry(
	i16_next_step:= , 
	i16_pos:= 2,
	s_debugtext:= ,
	E=> , 
	X=> , 
	i16_step=> ,
	i16_last_step=> );

fb_enum_find_file_list(
	sNetId:= '',
	sPathName:= ,
	eCmd:= ,
	pFindList:= ADR(arr_file_list),
	cbFindList:= SIZEOF(arr_file_list),
	bExecute:= ,
	tTimeout:= DEFAULT_ADS_TIMEOUT,
	bBusy=> ,
	bError=> ,
	nErrID=> , 
	bEOE=> ,
	nFindFiles=> );

fb_enum_find_file_entry(
	sNetId:= '',
	sPathName:= , 
	eCmd:= , 
	bExecute:= , 
	tTimeout:= DEFAULT_ADS_TIMEOUT,
	bBusy=> , 
	bError=> ,
	nErrID=> , 
	bEOE=> , 
	stFindFile=> );

fb_create_directory(
	sNetId:= '',
	sPathName:= ,
	ePath:= PATH_GENERIC,
	bExecute:= ,
	tTimeout:= DEFAULT_ADS_TIMEOUT,
	bBusy=> , 
	bError=> ,
	nErrId=> );

fb_file_open(
	sNetId:= '',
	sPathName:= , 
	nMode:= ,
	ePath:= PATH_GENERIC,
	bExecute:= , 
	tTimeout:= DEFAULT_ADS_TIMEOUT,
	bBusy=> , 
	bError=> , 
	nErrId=> , 
	hFile=> );

fb_file_close(
	sNetId:= '',
	hFile:= , 
	bExecute:= , 
	tTimeout:= t#10s,
	bBusy=> ,
	bError=> ,
	nErrId=> );

fb_file_write(
	sNetId:= '',
	hFile:= , 
	pWriteBuff:= ADR(temp_string),
	cbWriteLen:= LEN(temp_string),
	bExecute:= , 
	tTimeout:= t#10s,
	bBusy=> ,
	bError=> , 
	nErrId=> , 
	cbWrite=> );
END_FUNCTION_BLOCK

(* POU Gemeinsamkeiten17xx/XML Server/FB_Datei_erstellen, ST *)
FUNCTION_BLOCK FB_Datei_erstellen
VAR_INPUT
	bExecute					: BOOL;
	bQuit						: BOOL;
	s_path						: STRING;
	s_dateiname					: STRING;
	s_datei_erweiterung			: STRING;
	s_x_path_name				: STRING;
	s_symname					: STRING;
END_VAR
VAR_IN_OUT
END_VAR
VAR_OUTPUT
	bBusy						: BOOL;
	bError						: BOOL;
	nErrId						: UDINT;
END_VAR
VAR
	fb_enum_find_file_list			: FB_EnumFindFileList;
	fb_enum_find_file_entry			: FB_EnumFindFileEntry;
	fb_create_directory			: FB_CreateDir;	(* mit diesem FB kan nur eine Ordnerverzeichnissstruktur angelegt werden, jedoch keine Dateien erzeugt werden *)
	fb_file_open					: FB_FileOpen;	(* Eine vorhandene Datei öffnen oder eine Neue erzeugen *)
	fb_file_close					: FB_FileClose;
	fb_file_write					: FB_FileWrite;
	h_filehandle					: UINT := 0;(* file handle of the file *)
	arr_file_list					: ARRAY[0..63] OF ST_FindFileEntry;
	fb_ton_quitt					: TON;
	fb_r_trig_execute				: R_TRIG;
	fb_state_entry					: ST_StateEntry;
	temp_string					: STRING[255];
	i16_file_entry_zaehler			: INT := 0;
	i16_file_nr					: INT := 0;
	i							: INT := 0;
	b_pfad_vorhanden			: BOOL;
	b_datei_vorhanden			: BOOL;
END_VAR
fb_r_trig_execute(CLK:= bExecute, Q=> );
fb_ton_quitt(IN:= , PT:= t#100ms, Q=> , ET=> );

(* ======================================Schrittkette======================================== *)
fb_state_entry(
	i16_next_step:= ,
	i16_pos:= 1,
	s_debugtext:= ,
	E=> ,
	X=> ,
	i16_step=> ,
	i16_last_step=> );

CASE fb_state_entry.i16_step OF
(*=======================================================*)
	0:(* INIT *)
		bBusy := FALSE;
		bError := FALSE;
		nErrId := 0;
		fb_create_directory.bExecute := FALSE;
		fb_enum_find_file_list.bExecute := FALSE;
		fb_enum_find_file_entry.bExecute := FALSE;
		fb_file_open.bExecute := FALSE;
		fb_file_close.bExecute := FALSE;
		fb_state_entry.i16_next_step := 10;

(*=======================================================*)
	10:	(* Warte auf Execute-Befehl *)
		IF fb_state_entry.E THEN
			bBusy := FALSE;
		END_IF

		IF fb_r_trig_execute.Q THEN
			bBusy := TRUE;
			b_pfad_vorhanden := FALSE;
			b_datei_vorhanden := FALSE;
			fb_state_entry.i16_next_step := 20;
		END_IF

(*=======================================================*)
	20:	(* Prüfe, ob gewünschter Pfad auf dem Maschinen-PC vorhanden ist *)
		IF fb_state_entry.E THEN
			fb_enum_find_file_list.sPathName := s_path;
			fb_enum_find_file_list.eCmd := eEnumCmd_First;
			fb_enum_find_file_list.bExecute := TRUE;
		END_IF

		IF fb_enum_find_file_list.bBusy THEN
			fb_enum_find_file_list.bExecute := FALSE;
			fb_state_entry.i16_next_step := 30;
		END_IF

(*=======================================================*)
	30:	(* Auswerten des Ordner-Suchergebnis *)
		IF NOT fb_enum_find_file_list.bBusy THEN
			fb_enum_find_file_list.bExecute := FALSE;
		 	IF fb_enum_find_file_list.bError OR fb_enum_find_file_list.bEOE THEN
				 IF fb_enum_find_file_list.nFindFiles=0 THEN
					b_pfad_vorhanden := FALSE;
					fb_state_entry.i16_next_step := 40;	(* Pfad nicht vorhanden -> wird angelegt *)
				ELSE
					b_pfad_vorhanden := TRUE;
					fb_state_entry.i16_next_step := 60;	(* O.K. Pfad vorhanden -> Datei prüfen *)
				END_IF
			END_IF
		END_IF

(*=======================================================*)
	40:	(* Erstellen eines Ordnerverzeichnisses auf dem Laufwerk des Maschinen-PCs *)
		IF fb_state_entry.E THEN
			fb_create_directory.sPathName := s_path;
			fb_create_directory.bExecute := TRUE;
		END_IF

		IF fb_create_directory.bBusy THEN
			fb_create_directory.bExecute := FALSE;
			fb_state_entry.i16_next_step := 50;
		END_IF

(*=======================================================*)
	50:	(* Ordner wurde erstellt *)
		IF NOT fb_create_directory.bBusy  THEN
			IF NOT fb_create_directory.bError THEN
				fb_state_entry.i16_next_step := 60;	(* Ordnerverzeichnis wurde erfolgreich erstellt -> eine neue Datei anlegen oder eine Vorhandene öffnen *)
			ELSE
				fb_state_entry.i16_next_step := 1000;	(* Fehler *)
			END_IF
		END_IF

(*=======================================================*)
	60:	(* Prüfe, ob die gewünschte Datei in diesem Ordnerverzeichnis vorhanden ist *)
		IF fb_state_entry.E THEN
			temp_string := '';
			temp_string := CONCAT(temp_string, s_path);
			temp_string := CONCAT(temp_string, '\');
			temp_string := CONCAT(temp_string, s_dateiname);
			temp_string := CONCAT(temp_string, s_datei_erweiterung);
			fb_enum_find_file_entry.sPathName := temp_string;
			fb_enum_find_file_entry.eCmd := eEnumCmd_First;
			fb_enum_find_file_entry.bExecute := TRUE;
		END_IF

		IF fb_enum_find_file_entry.bBusy THEN
			fb_enum_find_file_entry.bExecute := FALSE;
			fb_state_entry.i16_next_step := 70;
		END_IF

(*=======================================================*)
	70:	(* Auswerten des Datei-Suchergebnis *)
		IF NOT fb_enum_find_file_entry.bBusy THEN
			fb_enum_find_file_entry.bExecute := FALSE;
		 	IF NOT fb_enum_find_file_entry.bError THEN
				IF fb_enum_find_file_entry.bEOE THEN
					IF fb_enum_find_file_entry.stFindFile.sFileName = CONCAT(s_dateiname, s_datei_erweiterung) THEN
					(* Datei bereits vorhanden *)
						b_datei_vorhanden := TRUE;
						fb_state_entry.i16_next_step := 0;
					ELSE
					(* Ende der Fileliste wurde erreicht und die gesuchte Datei ist  nicht vorhanden -> muss später angelegt werden *)
						b_datei_vorhanden := FALSE;
						fb_state_entry.i16_next_step := 100;
					END_IF
				ELSE
				(* Dateisuche im FB mit Abort korrekt beenden *)
					IF fb_enum_find_file_entry.stFindFile.sFileName = CONCAT(s_dateiname, s_datei_erweiterung) THEN
					(* Die gesuchte Datei wurde in der Fileliste gefunden *)
						b_datei_vorhanden := TRUE;
						fb_state_entry.i16_next_step := 80;
					ELSE
					(* Datei ist  nicht vorhanden -> muss später angelegt werden *)
						b_datei_vorhanden := FALSE;
						fb_state_entry.i16_next_step := 80;
					END_IF
				END_IF
			ELSE
				fb_state_entry.i16_next_step := FEHLER;
			END_IF
		END_IF

(*=======================================================*)
	80:	(* Dateisuchen wird beendet *)
		IF fb_state_entry.E THEN
			fb_enum_find_file_entry.eCmd := eEnumCmd_Abort;
			fb_enum_find_file_entry.bExecute := TRUE;
		END_IF

		IF fb_enum_find_file_entry.bBusy THEN
			fb_enum_find_file_entry.bExecute := FALSE;
			fb_state_entry.i16_next_step := 90;
		END_IF

(*=======================================================*)
	90:	(* Filehandle wieder frei *)
		IF NOT fb_enum_find_file_entry.bBusy THEN
			fb_enum_find_file_entry.bExecute := FALSE;
		 	IF NOT fb_enum_find_file_entry.bError AND fb_enum_find_file_entry.bEOE THEN
				fb_state_entry.i16_next_step := 100;
			ELSE
				fb_state_entry.i16_next_step := FEHLER;
			END_IF
		END_IF

(*=======================================================*)
	100:	(* Abfrage auf Datei anlegen *)
		IF fb_state_entry.E THEN
			IF NOT b_datei_vorhanden THEN
				fb_state_entry.i16_next_step := 110;
			ELSE
				fb_state_entry.i16_next_step := 0;	(* Fertig *)
			END_IF
		END_IF

(*=======================================================*)
	110:	(* Erzeugen einer neuen Datei *)
		IF fb_state_entry.E THEN
			temp_string := '';
			temp_string := CONCAT(temp_string, s_path);
			temp_string := CONCAT(temp_string, '\');
			temp_string := CONCAT(temp_string, s_dateiname);
			temp_string := CONCAT(temp_string, s_datei_erweiterung);
			fb_file_open.sPathName := temp_string;
			fb_file_open.nMode := FOPEN_MODEWRITE OR FOPEN_MODEBINARY;
			fb_file_open.bExecute := TRUE;
		END_IF

		IF fb_file_open.bBusy THEN
			fb_file_open.bExecute := FALSE;
			fb_state_entry.i16_next_step := 120;
		END_IF

(*=======================================================*)
	120:	(* Warte bis Datei geöffnet wurde *)
		IF NOT fb_file_open.bBusy  THEN
			IF NOT fb_file_open.bError THEN
				h_filehandle := fb_file_open.hFile;
				fb_state_entry.i16_next_step := 130;
			ELSE	(* Fehler *)
				nErrId := fb_file_open.nErrId;
				fb_state_entry.i16_next_step := 1000;
			END_IF
		END_IF

(*=======================================================*)
	130:	(* Schreibe die Dateistruktur im XML-Format: z.B.*)
		(*
		<Maschine1700_Datensicherung>
		<gst_datensatz>
		</gst_datensatz>
		</Maschine1700_Datensicherung>
		*)
		IF fb_state_entry.E THEN
			temp_string := '';
			temp_string := CONCAT(temp_string, '<');
			temp_string := CONCAT(temp_string, s_x_path_name);
			temp_string := CONCAT(temp_string, '>');
			temp_string := CONCAT(temp_string, '$r$n');

			(* Die Variable "s_xml_variablenname" wird hier schon mit angelegt, *)
			(* damit später beim "WECHSELN>" daraus gelesen werden kann, obwohl noch nichts drin steht *)
			temp_string := CONCAT(temp_string, '<');
			temp_string := CONCAT(temp_string, s_symname);
			temp_string := CONCAT(temp_string, '>');
			temp_string := CONCAT(temp_string, '$r$n');
			temp_string := CONCAT(temp_string, '<');
			temp_string := CONCAT(temp_string, '/');
			temp_string := CONCAT(temp_string, s_symname);
			temp_string := CONCAT(temp_string, '>');
			temp_string := CONCAT(temp_string, '$r$n');

			temp_string := CONCAT(temp_string, '<');
			temp_string := CONCAT(temp_string, '/');
			temp_string := CONCAT(temp_string, s_x_path_name);
			temp_string := CONCAT(temp_string, '>');
			fb_file_write.hFile := h_filehandle;
 			fb_file_write.bExecute := TRUE;
		END_IF

		IF fb_file_write.bBusy THEN
			fb_file_write.bExecute := FALSE;
			fb_state_entry.i16_next_step := 140;
		END_IF

(*=======================================================*)
	140:	(* Warte bis Datei geschrieben wurde *)
		IF NOT fb_file_write.bBusy  THEN
			IF NOT fb_file_write.bError THEN
				fb_state_entry.i16_next_step := 150;
			ELSE	(* Fehler *)
				nErrId := fb_file_write.nErrId;
				fb_state_entry.i16_next_step := 1000;
			END_IF
		END_IF

(*=======================================================*)
	150:	(* Schliesse Datei wieder, damit ein erneuter Zugriff möglich ist *)
		IF fb_state_entry.E THEN
			fb_file_close.hFile := h_filehandle;
			fb_file_close.bExecute := TRUE;
		END_IF

		IF fb_file_close.bBusy THEN
			fb_file_close.bExecute := FALSE;
			fb_state_entry.i16_next_step := 160;
		END_IF

(*=======================================================*)
	160:	(* Warte bis geschlossen *)
		IF NOT fb_file_close.bBusy  THEN
			IF NOT fb_file_close.bError THEN
				h_filehandle := 0;
				fb_state_entry.i16_next_step :=0;
			ELSE	(* Fehler *)
				nErrId := fb_file_close.nErrId;
				fb_state_entry.i16_next_step := 1000;
			END_IF
		END_IF

(*=======================================================*)
	1000: (* Fehler *)
		IF fb_state_entry.E THEN
			bBusy := FALSE;
			bError := TRUE;
			fb_ton_quitt.IN := FALSE;
		END_IF

		(*-----------------------Weiterschaltbedingungen----------------------------*)
		IF bQuit AND NOT fb_state_entry.E THEN
			bError := FALSE;
			fb_ton_quitt.IN := TRUE;
		END_IF

		IF fb_ton_quitt.Q THEN
			fb_ton_quitt.IN := FALSE;
			fb_state_entry.i16_next_step := 0;
		END_IF
END_CASE

fb_state_entry(
	i16_next_step:= , 
	i16_pos:= 2,
	s_debugtext:= ,
	E=> , 
	X=> , 
	i16_step=> ,
	i16_last_step=> );

fb_enum_find_file_list(
	sNetId:= '',
	sPathName:= ,
	eCmd:= ,
	pFindList:= ADR(arr_file_list),
	cbFindList:= SIZEOF(arr_file_list),
	bExecute:= ,
	tTimeout:= DEFAULT_ADS_TIMEOUT,
	bBusy=> ,
	bError=> ,
	nErrID=> , 
	bEOE=> ,
	nFindFiles=> );

fb_enum_find_file_entry(
	sNetId:= '',
	sPathName:= , 
	eCmd:= , 
	bExecute:= , 
	tTimeout:= DEFAULT_ADS_TIMEOUT,
	bBusy=> , 
	bError=> ,
	nErrID=> , 
	bEOE=> , 
	stFindFile=> );

fb_create_directory(
	sNetId:= '',
	sPathName:= ,
	ePath:= PATH_GENERIC,
	bExecute:= ,
	tTimeout:= DEFAULT_ADS_TIMEOUT,
	bBusy=> , 
	bError=> ,
	nErrId=> );

fb_file_open(
	sNetId:= '',
	sPathName:= , 
	nMode:= ,
	ePath:= PATH_GENERIC,
	bExecute:= , 
	tTimeout:= DEFAULT_ADS_TIMEOUT,
	bBusy=> , 
	bError=> , 
	nErrId=> , 
	hFile=> );

fb_file_close(
	sNetId:= '',
	hFile:= , 
	bExecute:= , 
	tTimeout:= t#10s,
	bBusy=> ,
	bError=> ,
	nErrId=> );

fb_file_write(
	sNetId:= '',
	hFile:= , 
	pWriteBuff:= ADR(temp_string),
	cbWriteLen:= LEN(temp_string),
	bExecute:= , 
	tTimeout:= t#10s,
	bBusy=> ,
	bError=> , 
	nErrId=> , 
	cbWrite=> );
END_FUNCTION_BLOCK

(* POU Gemeinsamkeiten17xx/XML Server/FB_XMLFileCopy, ST *)
FUNCTION_BLOCK FB_XMLFileCopy
VAR_INPUT
	srcNetId				: T_AmsNetId;	(* TwinCAT network address of the source file *)
	destNetId			: T_AmsNetId;	(* TwinCAT network address of the destination file *)
	bExecute			: BOOL;
	bQuit				: BOOL;
	s_name_quelldatei	: STRING;
	s_name_zieldatei		: STRING;
END_VAR
VAR_OUTPUT
	bBusy				: BOOL;
	bError				: BOOL;
	nErrId				: UDINT;
END_VAR
VAR
	fb_file_open			: FB_FileOpen;
	fb_file_close			: FB_FileClose;
	fb_file_read			: FB_FileRead;
	fb_file_write			: FB_FileWrite;

	h_quell_filehandle		: UINT := 0;(* file handle of the source file *)
	h_ziel_filehandle		: UINT := 0;(* file handle of the destination file *)

	fb_state_entry			: ST_StateEntry;
	fb_r_trig_execute		: R_TRIG;
	fb_ton_quitt			: TON;
	p_read_write_buffer	: ARRAY[1..100000] OF BYTE;
	cb_write_length		: UDINT :=0;
	cb_read_length		: UDINT :=0;
END_VAR
fb_r_trig_execute(CLK:= bExecute, Q=> );
fb_ton_quitt(IN:= , PT:= t#100ms, Q=> , ET=> );

(* ======================================Schrittkette======================================== *)
fb_state_entry(
	i16_next_step:= ,
	i16_pos:= 1,
	s_debugtext:= ,
	E=> ,
	X=> ,
	i16_step=> ,
	i16_last_step=> );

CASE fb_state_entry.i16_step OF
(*=======================================================*)
	0:(* INIT *)
		bBusy := FALSE;
		bError := FALSE;
		nErrId := 0;
		fb_file_open.bExecute := FALSE;
		fb_file_close.bExecute := FALSE;
		fb_file_read.bExecute := FALSE;
		fb_file_write.bExecute := FALSE;
		h_quell_filehandle := 0;
		h_ziel_filehandle := 0;
		cb_write_length :=0;
		cb_read_length :=0;
		fb_state_entry.i16_next_step := 10;

(*=======================================================*)
	10:	(* Warte auf Execute-Befehl *)
		IF fb_state_entry.E THEN
			bBusy := FALSE;
		END_IF

		IF fb_r_trig_execute.Q THEN
			bBusy := TRUE;
			fb_state_entry.i16_next_step := 100;
		END_IF

(*=======================================================*)
	100:	(* Öffne Quelldatei *)
		IF fb_state_entry.E THEN
			fb_file_open.nMode := FOPEN_MODEREAD OR FOPEN_MODEBINARY;
			fb_file_open.sPathName := s_name_quelldatei;
			fb_file_open.bExecute := TRUE;
		END_IF

		IF fb_file_open.bBusy THEN
			fb_file_open.bExecute := FALSE;
			fb_state_entry.i16_next_step := 110;
		END_IF

(*=======================================================*)
	110:	(* Warte bis Quelle geöffnet *)
		IF NOT fb_file_open.bBusy  THEN
			IF NOT fb_file_open.bError THEN
				h_quell_filehandle := fb_file_open.hFile;
				fb_state_entry.i16_next_step := 120;
			ELSE	(* Fehler *)
				nErrId := fb_file_open.nErrId;
				fb_state_entry.i16_next_step := 300;
			END_IF
		END_IF

(*=======================================================*)
	120:	(* Öffne Zieldatei *)
		IF fb_state_entry.E THEN
			fb_file_open.nMode := FOPEN_MODEWRITE OR FOPEN_MODEBINARY;
			fb_file_open.sPathName := s_name_zieldatei;
			fb_file_open.bExecute := TRUE;
		END_IF

		IF fb_file_open.bBusy THEN
			fb_file_open.bExecute := FALSE;
			fb_state_entry.i16_next_step := 130;
		END_IF

(*=======================================================*)
	130:	(* Warte bis Ziel geöffnet *)
		IF NOT fb_file_open.bBusy  THEN
			IF NOT fb_file_open.bError THEN
				h_ziel_filehandle := fb_file_open.hFile;
				fb_state_entry.i16_next_step := 150;
			ELSE	(* Fehler *)
				nErrId := fb_file_open.nErrId;
				fb_state_entry.i16_next_step := 300;
			END_IF
		END_IF

(*=======================================================*)
	150:	(* Lese Daten von der Quelldatei *)
		IF fb_state_entry.E THEN
			fb_file_read.hFile := h_quell_filehandle;
			fb_file_read.bExecute := TRUE;
		END_IF

		IF fb_file_read.bBusy THEN
			fb_file_read.bExecute := FALSE;
			fb_state_entry.i16_next_step := 160;
		END_IF

(*=======================================================*)
	160:	(* Warte bis gelesen *)
		IF NOT fb_file_read.bBusy  THEN
			IF NOT fb_file_read.bError THEN
				cb_read_length := fb_file_read.cbRead;
				fb_state_entry.i16_next_step := 170;
			ELSE	(* Fehler *)
				nErrId := fb_file_read.nErrId;
				fb_state_entry.i16_next_step := 300;
			END_IF
		END_IF

(*=======================================================*)
	170:	(* Schreibe Daten in die Zieldatei *)
		IF fb_state_entry.E THEN
			fb_file_write.hFile := h_ziel_filehandle;
			cb_write_length := cb_read_length;
			fb_file_write.bExecute := TRUE;
		END_IF

		IF fb_file_write.bBusy THEN
			fb_file_write.bExecute := FALSE;
			fb_state_entry.i16_next_step := 180;
		END_IF

(*=======================================================*)
	180:	(* Warte bis geschrieben *)
		IF NOT fb_file_write.bBusy  THEN
			IF NOT fb_file_write.bError THEN
				IF fb_file_read.bEOF THEN (* Prüfe, ob das EOF-Flag gesetzt ist *)
					fb_state_entry.i16_next_step := 200; (* Quell- und Zieldatei schliessen *)
				ELSE
					fb_state_entry.i16_next_step := 150; (* Weitere Daten lesen *)
				END_IF
			ELSE	(* Fehler *)
				nErrId := fb_file_write.nErrId;
				fb_state_entry.i16_next_step := 300;
			END_IF
		END_IF

(*=======================================================*)
	200:	(* Schliessen der Zieldatei *)
		IF fb_state_entry.E THEN
			fb_file_close.hFile := h_ziel_filehandle;
			fb_file_close.bExecute := TRUE;
		END_IF

		IF fb_file_close.bBusy THEN
			fb_file_close.bExecute := FALSE;
			fb_state_entry.i16_next_step := 210;
		END_IF

(*=======================================================*)
	210:	(* Warte bis Ziel geschlossen *)
		IF NOT fb_file_close.bBusy  THEN
			IF NOT fb_file_close.bError THEN
				h_ziel_filehandle := 0;
				fb_state_entry.i16_next_step := 220;
			ELSE	(* Fehler *)
				nErrId := fb_file_close.nErrId;
				fb_state_entry.i16_next_step := 300;
			END_IF
		END_IF

(*=======================================================*)
	220:	(* Schliessen der Quelldatei *)
		IF fb_state_entry.E THEN
			fb_file_close.hFile := h_quell_filehandle;
			fb_file_close.bExecute := TRUE;
		END_IF

		IF fb_file_close.bBusy THEN
			fb_file_close.bExecute := FALSE;
			fb_state_entry.i16_next_step := 230;
		END_IF

(*=======================================================*)
	230:	(* Warte bis Quelle geschlossen *)
		IF NOT fb_file_close.bBusy  THEN
			IF NOT fb_file_close.bError THEN
				h_quell_filehandle := 0;
				fb_state_entry.i16_next_step := 10;
			ELSE	(* Fehler *)
				nErrId := fb_file_close.nErrId;
				fb_state_entry.i16_next_step := 300;
			END_IF
		END_IF

(*=======================================================*)
	300:	(* Bei Fehler müssen Quell- und Zieldatei auf jeden Fall geschlossen werden *)
		(* Beide Dateien korrekt geschlossen -> Fehler auswerten *)
		IF ( h_ziel_filehandle = 0 AND h_quell_filehandle = 0 ) THEN
			fb_state_entry.i16_next_step := 1000;
		(* Beide Dateien sind noch offen und müsse zuerst geschlossen werden -> schliesse zuerst die Quelle*)
		ELSIF (h_quell_filehandle <> 0 AND h_ziel_filehandle <> 0 ) THEN
			fb_file_close.hFile := h_quell_filehandle;
			fb_state_entry.i16_next_step := 310;
		(* Quelle offen und Ziel geschlossen -> Quelle schliessen *)
		ELSIF (h_quell_filehandle <> 0 AND h_ziel_filehandle = 0 ) THEN
			fb_file_close.hFile := h_quell_filehandle;
			fb_state_entry.i16_next_step := 310; (* Schliesse Quelldatei *)
		(* Ziel offen und Quelle geschlossen -> Ziel schliessen *)
		ELSIF (h_quell_filehandle = 0 AND h_ziel_filehandle <> 0) THEN
			fb_file_close.hFile := h_ziel_filehandle;
			fb_state_entry.i16_next_step := 310; (* Schliesse Zielldatei *)
			bBusy := FALSE;
		END_IF

(*=======================================================*)
	310:	(* Schliessen der Datei *)
		IF fb_state_entry.E THEN
			fb_file_close.bExecute := TRUE;
		END_IF

		IF fb_file_close.bBusy THEN
			fb_file_close.bExecute := FALSE;
			fb_state_entry.i16_next_step := 320;
		END_IF

(*=======================================================*)
	320:	(* Warte bis geschlossen *)
		IF NOT fb_file_close.bBusy  THEN
			IF NOT fb_file_close.bError THEN
				IF fb_file_close.hFile = h_quell_filehandle THEN
					h_quell_filehandle := 0;
				ELSIF fb_file_close.hFile = h_ziel_filehandle THEN
					h_ziel_filehandle := 0;
				END_IF
				fb_state_entry.i16_next_step := 300;
			ELSE	(* Fehler *)
				nErrId := fb_file_close.nErrId;
				fb_state_entry.i16_next_step := 1000;
			END_IF
		END_IF

(*=======================================================*)
	1000: (* Fehler *)
		IF fb_state_entry.E THEN
			bBusy := FALSE;
			bError := TRUE;
			fb_ton_quitt.IN := FALSE;
		END_IF

		(*-----------------------Weiterschaltbedingungen----------------------------*)
		IF bQuit AND NOT fb_state_entry.E THEN
			bError := FALSE;
			fb_ton_quitt.IN := TRUE;
		END_IF

		IF fb_ton_quitt.Q THEN
			fb_ton_quitt.IN := FALSE;
			fb_state_entry.i16_next_step := 0;
		END_IF
END_CASE

fb_state_entry(
	i16_next_step:= , 
	i16_pos:= 2,
	s_debugtext:= ,
	E=> , 
	X=> , 
	i16_step=> ,
	i16_last_step=> );

fb_file_close(
	sNetId:= '',
	hFile:= , 
	bExecute:= , 
	tTimeout:= DEFAULT_ADS_TIMEOUT,
	bBusy=> ,
	bError=> , 
	nErrId=> );

fb_file_open(
	sNetId:= '',
	sPathName:= ,
	nMode:= 	,
	ePath:= PATH_GENERIC,
	bExecute:= , 
	tTimeout:= DEFAULT_ADS_TIMEOUT,
	bBusy=> ,
	bError=> , 
	nErrId=> ,
	hFile=> );

fb_file_read(
	sNetId:= ,
	hFile:= , 
	pReadBuff:= ADR(p_read_write_buffer),
	cbReadLen:= SIZEOF(p_read_write_buffer),
	bExecute:= , 
	tTimeout:= DEFAULT_ADS_TIMEOUT,
	bBusy=> , 
	bError=> ,
	nErrId=> ,
	cbRead=> , 
	bEOF=> );

fb_file_write(
	sNetId:= ,
	hFile:= ,
	pWriteBuff:= ADR(p_read_write_buffer),
	cbWriteLen:= cb_write_length,
	bExecute:= , 
	tTimeout:= DEFAULT_ADS_TIMEOUT,
	bBusy=> , 
	bError=> , 
	nErrId=> , 
	cbWrite=> );
END_FUNCTION_BLOCK
